(* IEC 61131-3 sources: POMIRTS_lab3/AS/Library_2/AsOpcUas, 3 files *)

(* ---- AsOpcUas.typ ---- *)
TYPE
	UaMethodOperateAction :
	(															(* Actions for UaSrv_MethodOperate		*)
    	UaMoa_CheckIsCalled 	:= 0,							(* Check if a method call is pending 	*)
	  	UaMoa_Finished         	:= 1							(* Finish method call					*)
	);
	UaSrv_MethodOperateInternal : STRUCT
		Busy					: BOOL;
		Execute					: BOOL;
		ModuleId				: UDINT;
		CallId					: UDINT;
		NamespaceIndex			: UINT;
		Reserved				: ARRAY[0..29] OF USINT;
	END_STRUCT;
	UaSrv_MethodCreateInternal : STRUCT
		Busy					: BOOL;
		Execute					: BOOL;
		ModuleId				: UDINT;
		Reserved				: ARRAY[0..31] OF USINT;
	END_STRUCT;
	UaSrv_MethodDeleteInternal : STRUCT
		Busy					: BOOL;
		Execute					: BOOL;
		ModuleId				: UDINT;
		Reserved				: ARRAY[0..31] OF USINT;
	END_STRUCT;
	UaSrv_FireEventInternal : STRUCT
		Busy					: BOOL;
		Execute					: BOOL;
		ModuleId				: UDINT;
		Reserved				: ARRAY[0..31] OF USINT;
	END_STRUCT;
	UaSrv_GetNamespaceIndexInternal : STRUCT
		Busy					: BOOL;
		Execute					: BOOL;
		ModuleId				: UDINT;
		Reserved				: ARRAY[0..31] OF USINT;
	END_STRUCT;
	UaSrv_DateTimeType : STRUCT
		DateTime				: DATE_AND_TIME;
		NanoSeconds				: UDINT;
	END_STRUCT;
	UaSrv_FireEventFieldType : STRUCT
		BrowsePath				: STRING[MAX_LENGTH_EVENTFIELDPATH];
		Variable				: STRING[MAX_LENGTH_VARIABLE];
		ErrorID					: DWORD;
	END_STRUCT;
END_TYPE

(* ---- AsOpcUas.fun ---- *)
FUNCTION_BLOCK UaSrv_MethodOperate
	VAR_INPUT
		Execute	           		: BOOL;
		MethodName				: STRING[255];
		Action					: UaMethodOperateAction;
	END_VAR

	VAR_OUTPUT
		IsCalled      			: BOOL;
		Done			   		: BOOL;
		Busy               		: BOOL;
		Error              		: BOOL;
		ErrorID            		: DWORD;
	END_VAR

	VAR
		Internal				: UaSrv_MethodOperateInternal;
	END_VAR
END_FUNCTION_BLOCK

FUNCTION_BLOCK UaSrv_MethodCreate
	VAR_INPUT
		Execute	           		: BOOL;
		MethodName				: STRING[255];
		InputArguments			: ARRAY[0..9] OF UAMethodArgument;
		OutputArguments			: ARRAY[0..9] OF UAMethodArgument;
	END_VAR

	VAR_OUTPUT
		Done			   		: BOOL;
		Busy               		: BOOL;
		Error              		: BOOL;
		ErrorID            		: DWORD;
	END_VAR

	VAR
		Internal				: UaSrv_MethodCreateInternal;
	END_VAR
END_FUNCTION_BLOCK

FUNCTION_BLOCK UaSrv_MethodDelete
	VAR_INPUT
		Execute	           		: BOOL;
		MethodName				: STRING[255];
	END_VAR

	VAR_OUTPUT
		Done			   		: BOOL;
		Busy               		: BOOL;
		Error              		: BOOL;
		ErrorID            		: DWORD;
	END_VAR

	VAR
		Internal				: UaSrv_MethodDeleteInternal;
	END_VAR
END_FUNCTION_BLOCK

FUNCTION_BLOCK UaSrv_GetNamespaceIndex
	VAR_INPUT
		Execute	           		: BOOL;
		NamespaceUri			: STRING[MAX_LENGTH_NAMESPACEURI];
	END_VAR

	VAR_OUTPUT
		NamespaceIndex			: UINT;
		Done			   		: BOOL;
		Busy               		: BOOL;
		Error              		: BOOL;
		ErrorID            		: DWORD;
	END_VAR

	VAR
		Internal				: UaSrv_GetNamespaceIndexInternal;
	END_VAR
END_FUNCTION_BLOCK

FUNCTION_BLOCK UaSrv_FireEvent
	VAR_INPUT
		Execute	           		: BOOL;
		EventType				: UANodeID;
		EventFieldCount			: UINT;
	END_VAR

	VAR_OUTPUT
		Done			   		: BOOL;
		Busy               		: BOOL;
		Error              		: BOOL;
		ErrorID            		: DWORD;
	END_VAR

	VAR_IN_OUT
		EventFields				: UaSrv_FireEventFieldType;
	END_VAR

	VAR
		Internal				: UaSrv_FireEventInternal;
	END_VAR
END_FUNCTION_BLOCK

(* ---- AsOpcUas.var ---- *)
VAR CONSTANT
	MAX_LENGTH_EVENTFIELDPATH			: UINT := 255;
	MAX_LENGTH_NAMESPACEURI				: UINT := 255;
END_VAR
